(* Logix 5000 project; controller IF2_DEMO Emulate 5570 rev 20.12; software revision 20.04; part 7 of 8 *)
(* tags used below, declared in another part *)
   Alarm_Packer1_Blocked : ALARM_DIGITAL;
   Alarm_Packer1_Starved : ALARM_DIGITAL;
   Alarm_Packer1_Stopped : ALARM_DIGITAL;
   Current_OEE_Availability : REAL;
   Current_OEE_Availability_MUL100 : DINT;
   Current_OEE_Available : REAL;
   Current_OEE_AvailableTimer : TIMER;
   Current_OEE_Overall : REAL;
   Current_OEE_Performance : REAL;
   Current_OEE_Performance_MUL100 : DINT;
   Current_OEE_Quality : REAL;
   Current_OEE_Quality_MUL100 : DINT;
   Current_OEE_Running : REAL;
   Current_OEE_RunningTimer : TIMER;
   OEE_Availability_Previous_1 : REAL;
   OEE_Availability_Previous_2 : REAL;
   OEE_Availability_Previous_3 : REAL;
   OEE_Overall_Previous_1 : REAL;
   OEE_Overall_Previous_2 : REAL;
   OEE_Overall_Previous_3 : REAL;
   OEE_Performance_Previous_1 : REAL;
   OEE_Performance_Previous_2 : REAL;
   OEE_Performance_Previous_3 : REAL;
   OEE_Quality_Previous_1 : REAL;
   OEE_Quality_Previous_2 : REAL;
   OEE_Quality_Previous_3 : REAL;
   OutputTargetTimer : TIMER;
   Packaging_Cases_Good : DINT;
   Packaging_Cases_Per_Minute : REAL;
   Packaging_Cases_Rejected : DINT;
   Packaging_Cases_Total : DINT;
   Packaging_Status : DINT;
   Packer : FTVPDemoWorkCell;
   Packer_State : DINT;
   TempReadTrigger : TIMER;
   TempTimer : TIMER;
   TempTimer2 : TIMER;
   ChangeOver_In_Progress : BOOL;
   Current_Order : STRING;
   CurrentCustomerName : STRING;
   CurrentPartName : STRING;
   IF_OEE : IF_OEE;
   InstantFizz_Plant : Plant;
   Line1 : FTVPDemoLine;
   Line_State_String : State;
   LineStates : STRING[4];
   NewOrder_Trigger : Event_Triggers;
   OEE_Part_Scrap_Old : DINT;
   OEE_Parts_Good_Old : DINT;
   OEE_Parts_Total_Old : DINT;
   OEE_Scrap_Filler : DINT;
   OEE_Scrap_Labeler : DINT;
   OEE_Scrap_Packaging : DINT;
   OrderQty : DINT[4];
   PartCountRollOver : DINT;
   Performance_Control : DINT;
   Previous_Order : STRING;
   PreviousCustomerName : STRING;
   PreviousPartName : STRING;
   ProdCounts : Counts;
   Timer1000ms : TIMER;
   Timer250ms : TIMER;
   WallClock : DINT[7];
   WC : WC[10];
(* PackD, continued *)

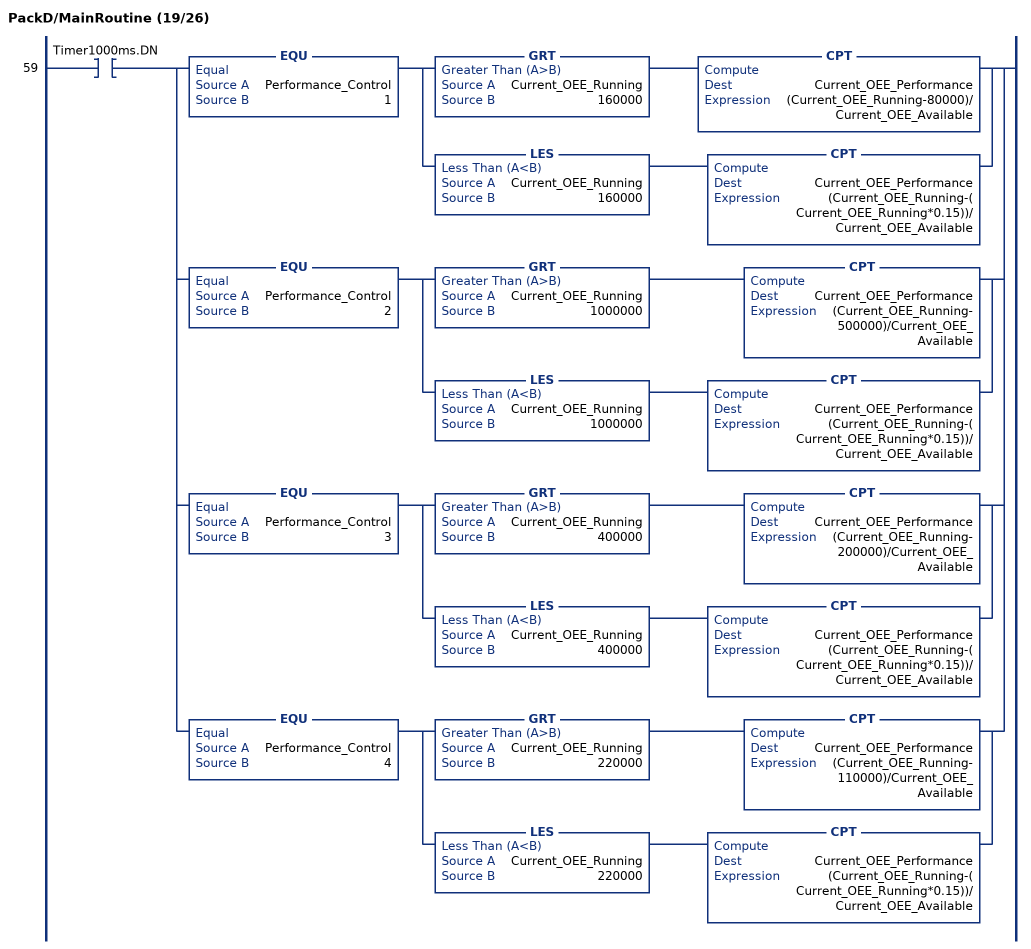
   59: XIC(Timer1000ms.DN)[EQU(Performance_Control,1) [GRT(Current_OEE_Running,160000) CPT(Current_OEE_Performance,(Current_OEE_Running-80000)/Current_OEE_Available) ,LES(Current_OEE_Running,160000) CPT(Current_OEE_Performance,(Current_OEE_Running-(Current_OEE_Running*0.15))/Current_OEE_Available) ] ,EQU(Performance_Control,2) [GRT(Current_OEE_Running,1000000) CPT(Current_OEE_Performance,(Current_OEE_Running-500000)/Current_OEE_Available) ,LES(Current_OEE_Running,1000000) CPT(Current_OEE_Performance,(Current_OEE_Running-(Current_OEE_Running*0.15))/Current_OEE_Available) ] ,EQU(Performance_Control,3) [GRT(Current_OEE_Running,400000) CPT(Current_OEE_Performance,(Current_OEE_Running-200000)/Current_OEE_Available) ,LES(Current_OEE_Running,400000) CPT(Current_OEE_Performance,(Current_OEE_Running-(Current_OEE_Running*0.15))/Current_OEE_Available) ] ,EQU(Performance_Control,4) [GRT(Current_OEE_Running,220000) CPT(Current_OEE_Performance,(Current_OEE_Running-110000)/Current_OEE_Available) ,LES(Current_OEE_Running,220000) CPT(Current_OEE_Performance,(Current_OEE_Running-(Current_OEE_Running*0.15))/Current_OEE_Available) ] ];
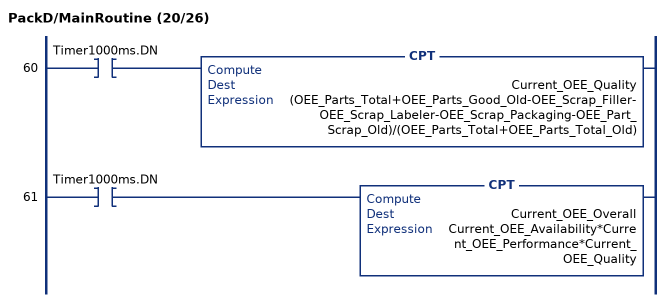
   60: XIC(Timer1000ms.DN)CPT(Current_OEE_Quality,(OEE_Parts_Total+OEE_Parts_Good_Old-OEE_Scrap_Filler-OEE_Scrap_Labeler-OEE_Scrap_Packaging-OEE_Part_Scrap_Old)/(OEE_Parts_Total+OEE_Parts_Total_Old));
   61: XIC(Timer1000ms.DN)CPT(Current_OEE_Overall,Current_OEE_Availability*Current_OEE_Performance*Current_OEE_Quality);
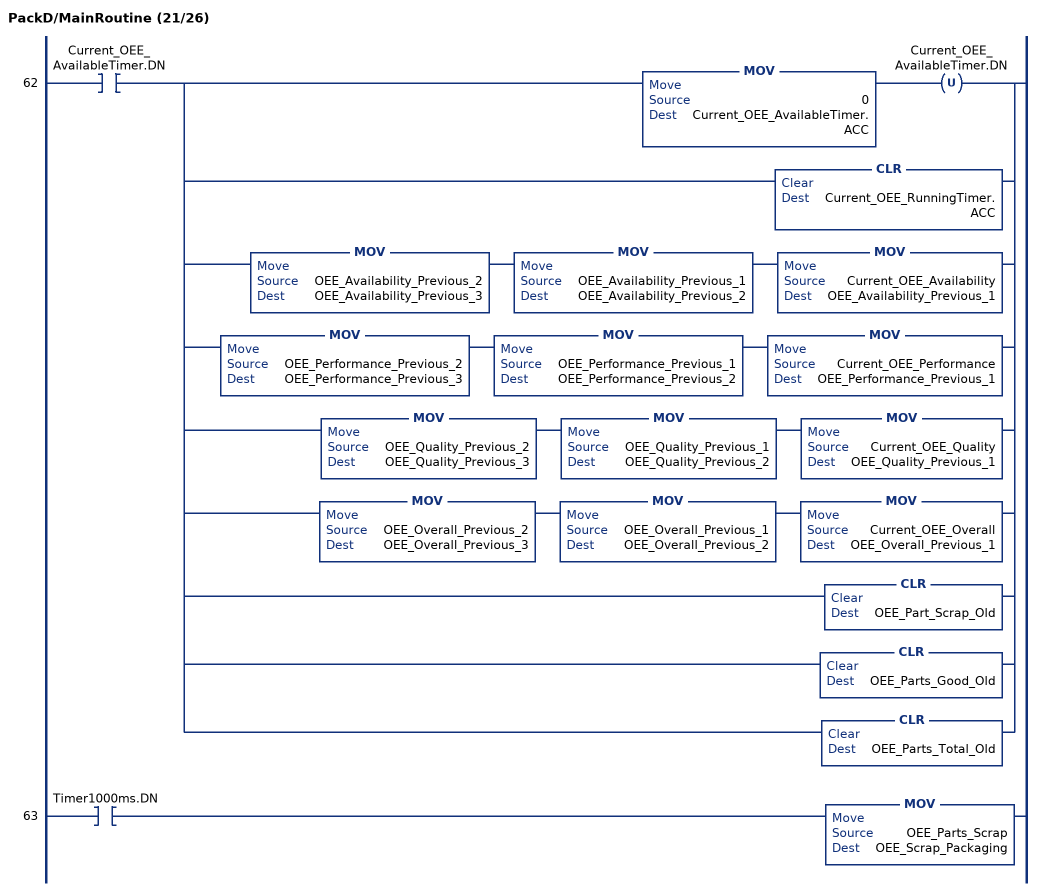
   62: XIC(Current_OEE_AvailableTimer.DN)[MOV(0,Current_OEE_AvailableTimer.ACC) OTU(Current_OEE_AvailableTimer.DN) ,CLR(Current_OEE_RunningTimer.ACC) ,MOV(OEE_Availability_Previous_2,OEE_Availability_Previous_3) MOV(OEE_Availability_Previous_1,OEE_Availability_Previous_2) MOV(Current_OEE_Availability,OEE_Availability_Previous_1) ,MOV(OEE_Performance_Previous_2,OEE_Performance_Previous_3) MOV(OEE_Performance_Previous_1,OEE_Performance_Previous_2) MOV(Current_OEE_Performance,OEE_Performance_Previous_1) ,MOV(OEE_Quality_Previous_2,OEE_Quality_Previous_3) MOV(OEE_Quality_Previous_1,OEE_Quality_Previous_2) MOV(Current_OEE_Quality,OEE_Quality_Previous_1) ,MOV(OEE_Overall_Previous_2,OEE_Overall_Previous_3) MOV(OEE_Overall_Previous_1,OEE_Overall_Previous_2) MOV(Current_OEE_Overall,OEE_Overall_Previous_1) ,CLR(OEE_Part_Scrap_Old) ,CLR(OEE_Parts_Good_Old) ,CLR(OEE_Parts_Total_Old) ];
   63: XIC(Timer1000ms.DN)MOV(OEE_Parts_Scrap,OEE_Scrap_Packaging);
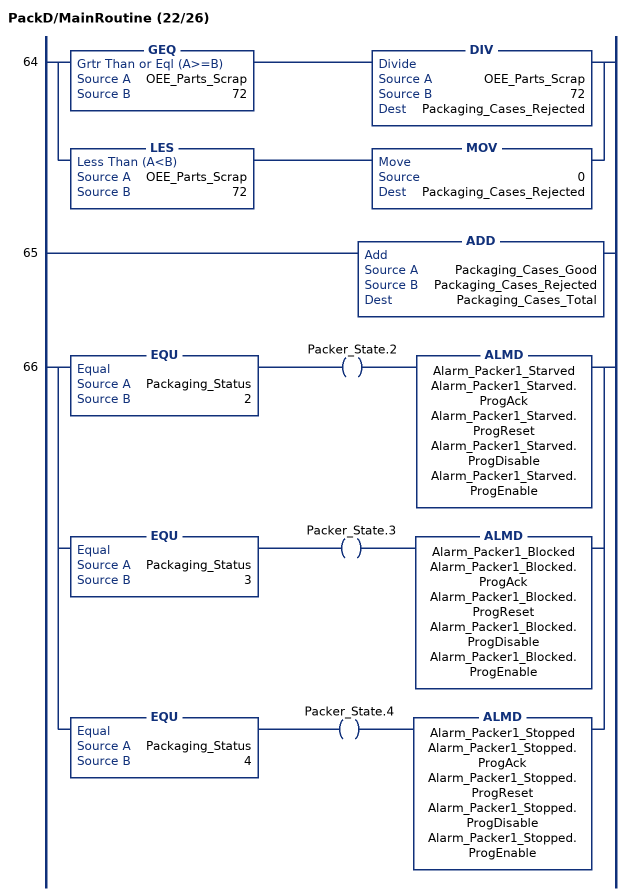
   64: [GEQ(OEE_Parts_Scrap,72) DIV(OEE_Parts_Scrap,72,Packaging_Cases_Rejected) ,LES(OEE_Parts_Scrap,72) MOV(0,Packaging_Cases_Rejected) ];
   65: ADD(Packaging_Cases_Good,Packaging_Cases_Rejected,Packaging_Cases_Total);
   66: [EQU(Packaging_Status,2) OTE(Packer_State.2) ALMD(Alarm_Packer1_Starved,Alarm_Packer1_Starved.ProgAck,Alarm_Packer1_Starved.ProgReset,Alarm_Packer1_Starved.ProgDisable,Alarm_Packer1_Starved.ProgEnable) ,EQU(Packaging_Status,3) OTE(Packer_State.3) ALMD(Alarm_Packer1_Blocked,Alarm_Packer1_Blocked.ProgAck,Alarm_Packer1_Blocked.ProgReset,Alarm_Packer1_Blocked.ProgDisable,Alarm_Packer1_Blocked.ProgEnable) ,EQU(Packaging_Status,4) OTE(Packer_State.4) ALMD(Alarm_Packer1_Stopped,Alarm_Packer1_Stopped.ProgAck,Alarm_Packer1_Stopped.ProgReset,Alarm_Packer1_Stopped.ProgDisable,Alarm_Packer1_Stopped.ProgEnable) ];
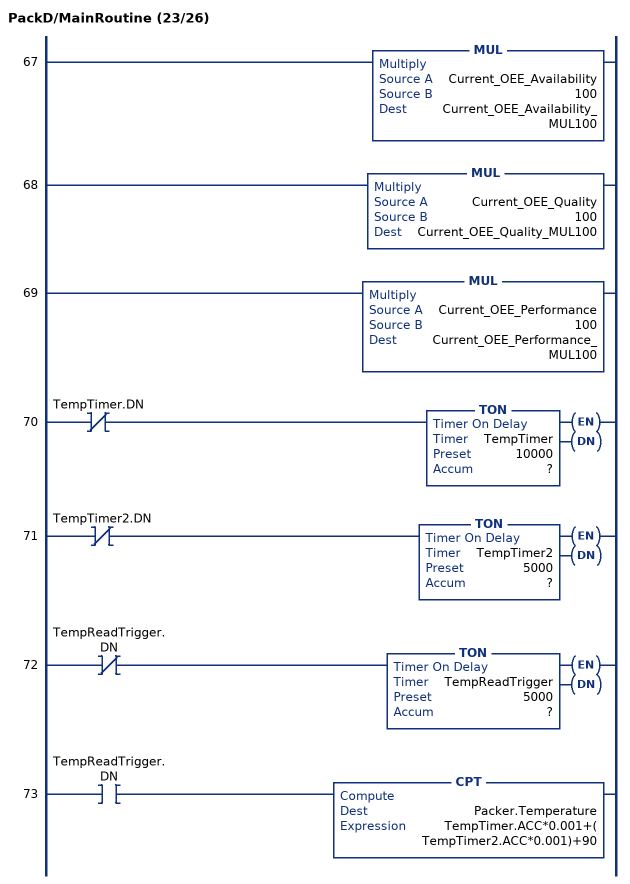
   67: MUL(Current_OEE_Availability,100,Current_OEE_Availability_MUL100);
   68: MUL(Current_OEE_Quality,100,Current_OEE_Quality_MUL100);
   69: MUL(Current_OEE_Performance,100,Current_OEE_Performance_MUL100);
   70: XIO(TempTimer.DN)TON(TempTimer,?,?);
   71: XIO(TempTimer2.DN)TON(TempTimer2,?,?);
   72: XIO(TempReadTrigger.DN)TON(TempReadTrigger,?,?);
   73: XIC(TempReadTrigger.DN)CPT(Packer.Temperature,TempTimer.ACC*0.001+(TempTimer2.ACC*0.001)+90);
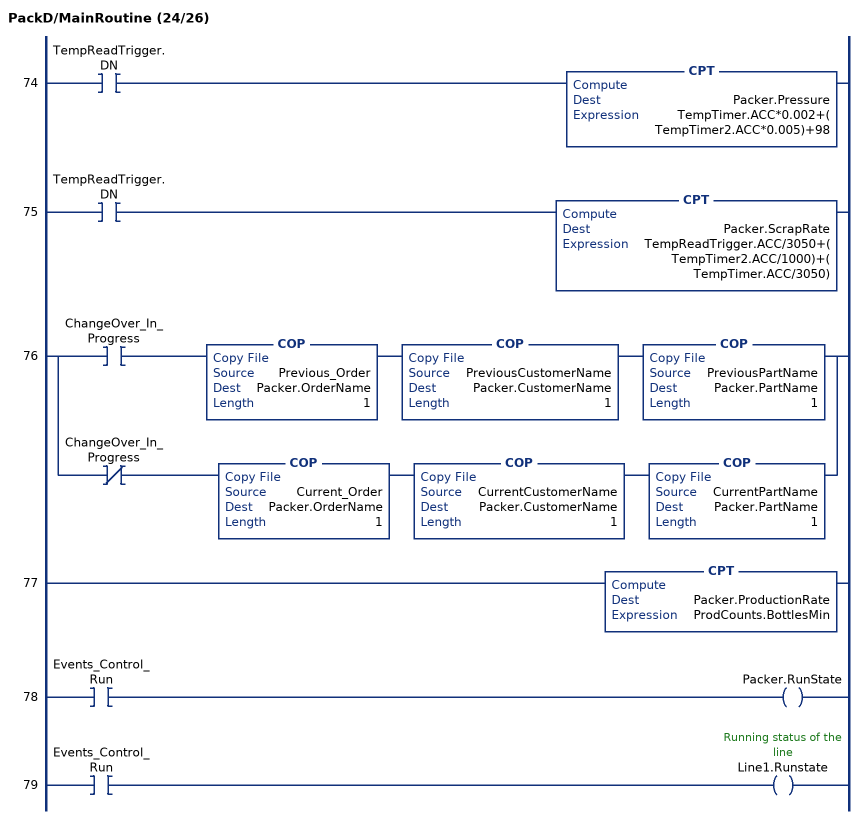
   74: XIC(TempReadTrigger.DN)CPT(Packer.Pressure,TempTimer.ACC*0.002+(TempTimer2.ACC*0.005)+98);
   75: XIC(TempReadTrigger.DN)CPT(Packer.ScrapRate,TempReadTrigger.ACC/3050+(TempTimer2.ACC/1000)+(TempTimer.ACC/3050));
   76: [XIC(ChangeOver_In_Progress) COP(Previous_Order,Packer.OrderName,1) COP(PreviousCustomerName,Packer.CustomerName,1) COP(PreviousPartName,Packer.PartName,1) ,XIO(ChangeOver_In_Progress) COP(Current_Order,Packer.OrderName,1) COP(CurrentCustomerName,Packer.CustomerName,1) COP(CurrentPartName,Packer.PartName,1) ];
   77: CPT(Packer.ProductionRate,ProdCounts.BottlesMin);
   78: XIC(Events_Control_Run)OTE(Packer.RunState);
   79: XIC(Events_Control_Run)OTE(Line1.Runstate);
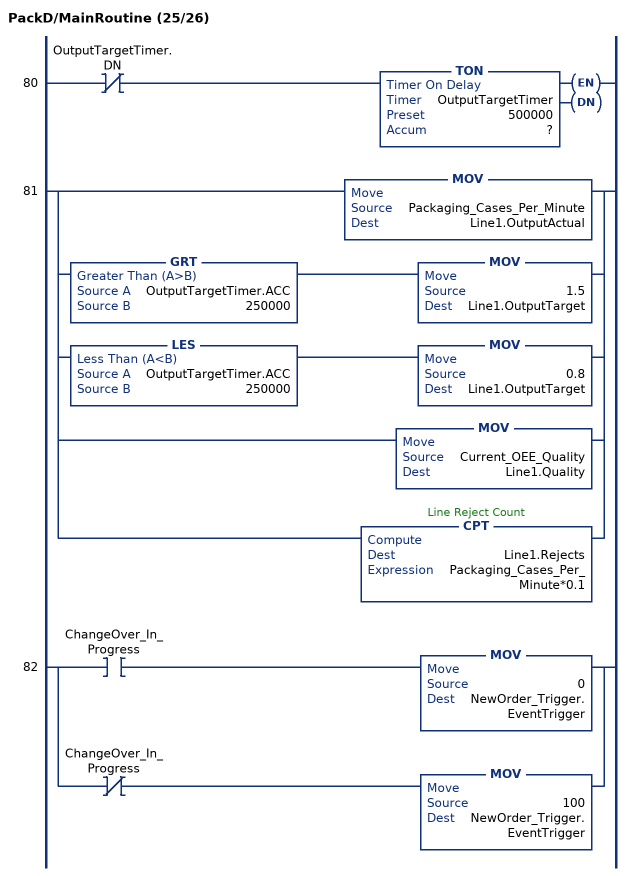
   80: XIO(OutputTargetTimer.DN)TON(OutputTargetTimer,?,?);
   81: [MOV(Packaging_Cases_Per_Minute,Line1.OutputActual) ,[GRT(OutputTargetTimer.ACC,250000) MOV(1.5,Line1.OutputTarget) ,LES(OutputTargetTimer.ACC,250000) MOV(0.8,Line1.OutputTarget) ] ,MOV(Current_OEE_Quality,Line1.Quality) ,CPT(Line1.Rejects,Packaging_Cases_Per_Minute*0.1) ];
   82: [XIC(ChangeOver_In_Progress) MOV(0,NewOrder_Trigger.EventTrigger) ,XIO(ChangeOver_In_Progress) MOV(100,NewOrder_Trigger.EventTrigger) ];
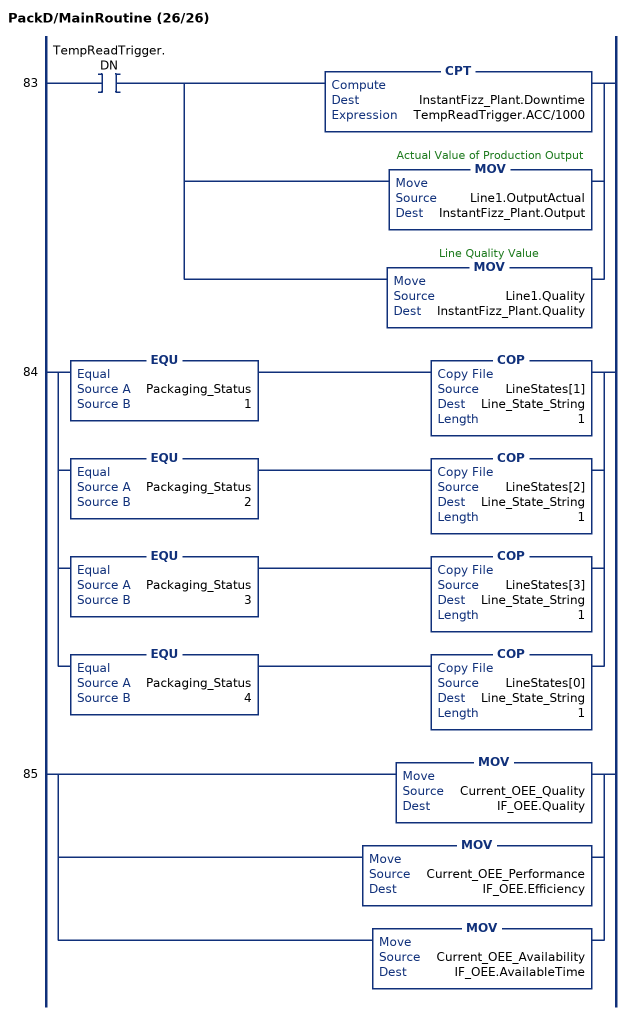
   83: XIC(TempReadTrigger.DN)[CPT(InstantFizz_Plant.Downtime,TempReadTrigger.ACC/1000) ,MOV(Line1.OutputActual,InstantFizz_Plant.Output) ,MOV(Line1.Quality,InstantFizz_Plant.Quality) ];
   84: [EQU(Packaging_Status,1) COP(LineStates[1],Line_State_String,1) ,EQU(Packaging_Status,2) COP(LineStates[2],Line_State_String,1) ,EQU(Packaging_Status,3) COP(LineStates[3],Line_State_String,1) ,EQU(Packaging_Status,4) COP(LineStates[0],Line_State_String,1) ];
   85: [MOV(Current_OEE_Quality,IF_OEE.Quality) ,MOV(Current_OEE_Performance,IF_OEE.Efficiency) ,MOV(Current_OEE_Availability,IF_OEE.AvailableTime) ];
END_ROUTINE
END_PROGRAM

PROGRAM Packer1   (* main routine MainRoutine *)
VAR
   Auto_setpoint : DINT := 3;
   Blinker : TIMER := (PRE := 1000, ACC := 931, EN := 1, TT := 1);
   Blocked_L : BOOL;
   Bottle_count_switch : BOOL := 1;
   Bottle_Counter : COUNTER := (ACC := 5098, CU := 1, DN := 1);
   BTank1_heat_ON : BOOL := 1;   // start heating
   BTank2_heat_ON : BOOL := 1;
   BTank3_heat_ON : BOOL := 1;
   BTMTimer_BTank1 : TIMER := (PRE := 1, EN := 1, TT := 1);   // Batch Tank1 timer
        .DN   // Batch Tank1 timer
   BTMTimer_BTank2 : TIMER := (PRE := 1, EN := 1, TT := 1);
   BTMTimer_BTank3 : TIMER := (PRE := 1, EN := 1, TT := 1);
   Drive_running : BOOL := 1;
   E_Stop : BOOL := 1;
   Events : Events := (Operate.OrderProc := 1, Control.StandbyCode := 3);
   Events_Control_Auto : ALIAS FOR WC_L.EventTrigger[0].5;
   Events_Control_Run : ALIAS FOR WC_L.EventTrigger[0].1;
   Events_Control_Standby : ALIAS FOR WC_L.EventTrigger[0].0;
   Events_Control_StandbyCode : ALIAS FOR WC_L.EventValue_REAL[1];
   Events_DownTime_Breakdown : ALIAS FOR WC_L.EventTrigger[0].2;
   Events_DownTime_BreakdownCode : ALIAS FOR WC_L.EventValue_REAL[2];
   Events_DownTime_Testing : ALIAS FOR WC_L.EventTrigger[0].7;
   Events_DownTime_UnschedMaint : ALIAS FOR WC_L.EventTrigger[0].6;
   Events_Operate_Load : ALIAS FOR WC_L.EventTrigger[0].10;
   Events_Operate_OrderProc : ALIAS FOR WC_L.EventTrigger[0].11;
   Events_Operate_Setup : ALIAS FOR WC_L.EventTrigger[0].9;
   Fill1_pressure : DINT := 150;   // Batch Tank1 pressure
   Fill2_pressure : DINT := 32;
   Fill3_pressure : DINT := 21;
   Heat_rate1 : REAL := 0.0003;   // value between 0 and 0.1
   Heat_rate2 : REAL := 0.0007;
   Heat_rate3 : REAL := 1.e-04;
   HMI : HMIVars := (ScrapRate := 5.0, SpeedControl := 100.0, PrevSpeed := 100.0, PartCountRollOver := 9999999, MfgTimeBase := 1, MaxEventDur := 19.0, MinEventDur := 6.0, EventsPerHr := 100, EventDur := 9.167803, RunDur := 25.832197, MinRunDur := 5.0);
   Jog : BOOL;
   Jog_PB : BOOL;
   Manual : BOOL;
   MaxPsiSP1 : DINT := 150;   // maximum pressure setpoint
   MaxPsiSP2 : DINT := 150;
   MaxPsiSP3 : DINT := 150;
   MaxTempSP1 : DINT := 220;   // maximum temperature set point
   MaxTempSP2 : DINT := 220;
   MaxTempSP3 : DINT := 220;
   MfgOrders : MfgOrders := (CustomerName := 'MRP', OrderName := 'Product B 1', GetNextOrder := 1, OrderQty := 600, ProdRate := 11.0, SetupTime := 8.0, PartName := 'Bottle3', WorkcellName := 'Capper 3', OperationId := 1006558);
   MfgOrders_CustomerName : ALIAS FOR WC_L.FlexSTRING[4];
   MfgOrders_OrderName : ALIAS FOR WC_L.FlexSTRING[3];
   MfgOrders_PartName : ALIAS FOR WC_L.FlexSTRING[0];
   MinPsiSP1 : DINT;   // minimum pressure setpoint
   MinPsiSP2 : DINT;
   MinPsiSP3 : DINT;
   MinTempSP1 : DINT := 60;   // minimum setpoint for temperature
   MinTempSP2 : DINT := 60;
   MinTempSP3 : DINT := 60;
   Motor1_temperature : DINT := 220;   // Motor1Temperature
   Motor2_temperature : DINT := 101;
   Motor3_temperature : DINT := 77;
   OEE : OEE := (IdealCycleTime := 5.0);
   OEE_IdealCycleTime : ALIAS FOR WC_L.IdealCT;
   OEE_Parts_Good : ALIAS FOR WC_L.GoodParts;
   OEE_Parts_Scrap : ALIAS FOR WC_L.ScrapParts;
   OEE_Parts_Total : ALIAS FOR WC_L.TotalParts;
   Run_PB : BOOL;
   Run_PL : BOOL := 1;
   Run_start_timer : TIMER := (PRE := 2000);
   Running : BOOL := 1;
   SIM : SimVars := (Run.PRE := 25832, Event.PRE := 9168, Setup.PRE := 6000, EventNumber := 7, UtilityBool[2] := 1);
        .UTILITYBOOL[2]   // First Scan Bit
   Sin_input_float1 : REAL := 1.667488;
   Sin_input_float2 : REAL := 5.7742753;
   Sin_input_float3 : REAL := 4.0464277;
   Speed_setpoint : DINT := 3;
   Starved_L : BOOL;
   Stop_PB : BOOL;
   Stop_PL : BOOL;
   Suppress : Events;
   WC_L : ALIAS FOR WC[6];
END_VAR

ROUTINE MainRoutine   (* ladder *)
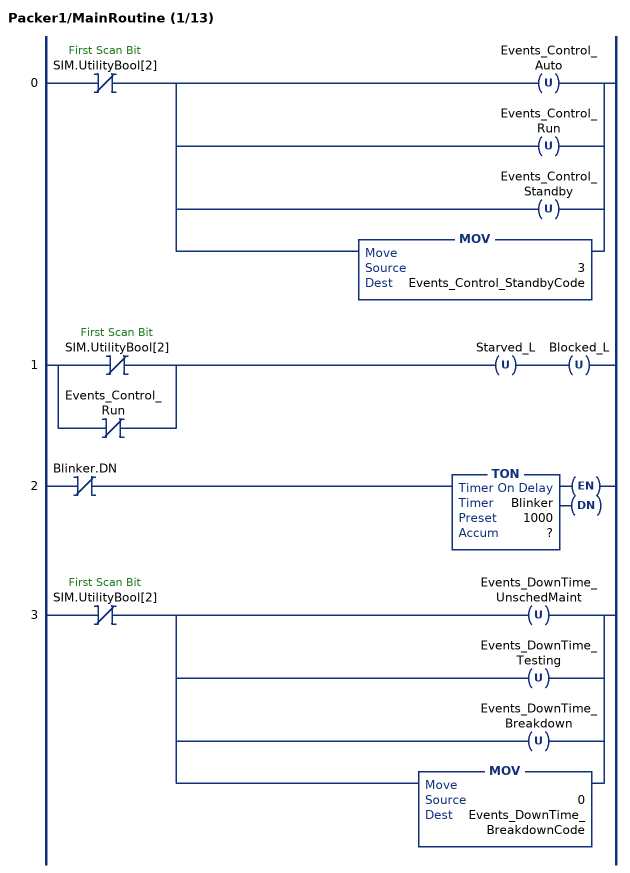
   0: XIO(SIM.UtilityBool[2])[OTU(Events_Control_Auto) ,OTU(Events_Control_Run) ,OTU(Events_Control_Standby) ,MOV(3,Events_Control_StandbyCode) ];
   1: [XIO(SIM.UtilityBool[2]) ,XIO(Events_Control_Run) ]OTU(Starved_L)OTU(Blocked_L);
   2: XIO(Blinker.DN)TON(Blinker,?,?);
   3: XIO(SIM.UtilityBool[2])[OTU(Events_DownTime_UnschedMaint) ,OTU(Events_DownTime_Testing) ,OTU(Events_DownTime_Breakdown) ,MOV(0,Events_DownTime_BreakdownCode) ];
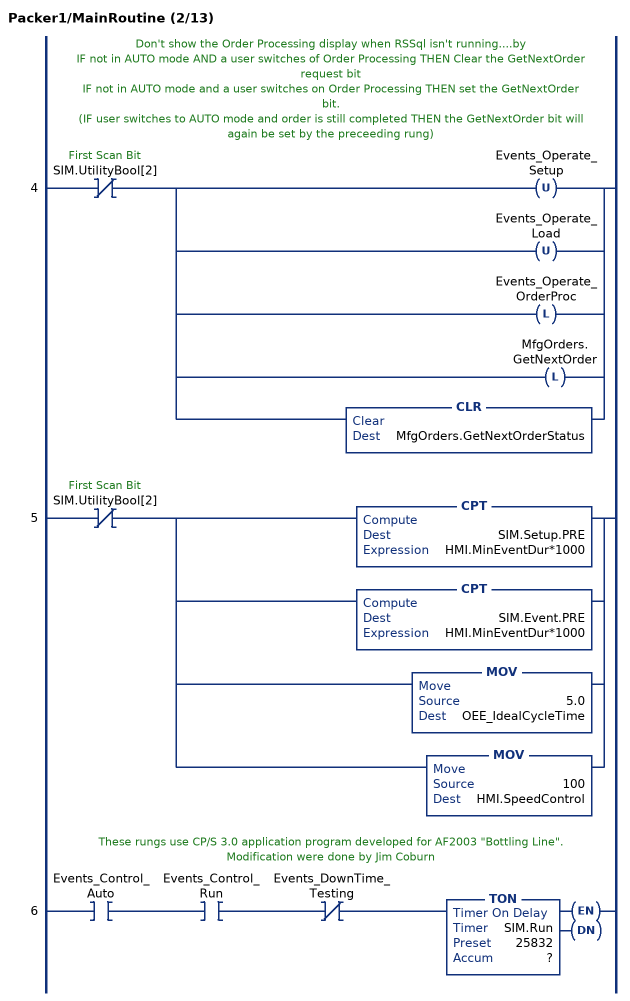
   // Don't show the Order Processing display when RSSql isn't running....by
   // IF not in AUTO mode AND a user switches of Order Processing THEN Clear the GetNextOrder request bit
   // IF not in AUTO mode and a user switches on Order Processing THEN set the GetNextOrder bit.
   // (IF user switches to AUTO mode and order is still completed THEN the GetNextOrder bit will again be set by the preceeding rung)
   4: XIO(SIM.UtilityBool[2])[OTU(Events_Operate_Setup) ,OTU(Events_Operate_Load) ,OTL(Events_Operate_OrderProc) ,OTL(MfgOrders.GetNextOrder) ,CLR(MfgOrders.GetNextOrderStatus) ];
   5: XIO(SIM.UtilityBool[2])[CPT(SIM.Setup.PRE,HMI.MinEventDur*1000) ,CPT(SIM.Event.PRE,HMI.MinEventDur*1000) ,MOV(5.0,OEE_IdealCycleTime) ,MOV(100,HMI.SpeedControl) ];
   // These rungs use CP/S 3.0 application program developed for AF2003 "Bottling Line".
   // Modification were done by Jim Coburn
   6: XIC(Events_Control_Auto)XIC(Events_Control_Run)XIO(Events_DownTime_Testing)TON(SIM.Run,?,?);
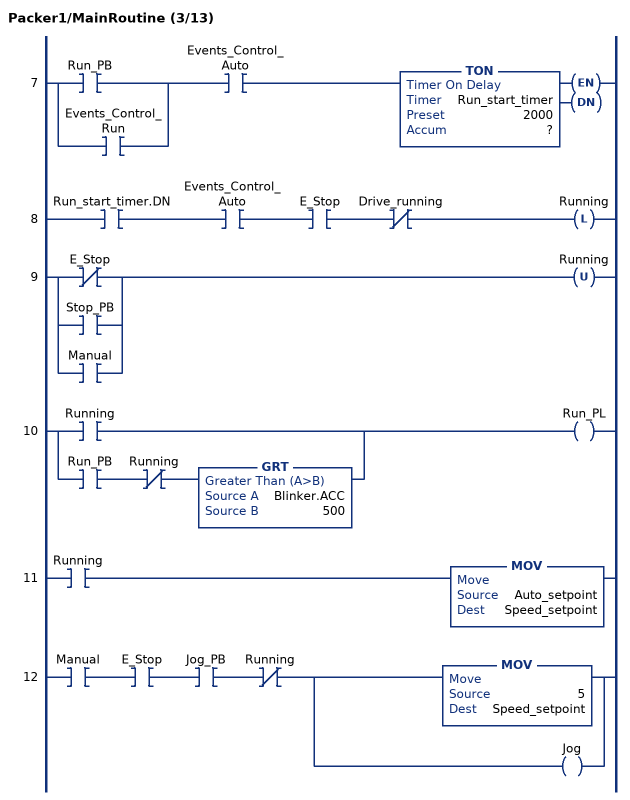
   7: [XIC(Run_PB) ,XIC(Events_Control_Run) ]XIC(Events_Control_Auto)TON(Run_start_timer,?,?);
   8: XIC(Run_start_timer.DN)XIC(Events_Control_Auto)XIC(E_Stop)XIO(Drive_running)OTL(Running);
   9: [XIO(E_Stop) ,[XIC(Stop_PB) ,XIC(Manual) ] ]OTU(Running);
   10: [XIC(Running) ,XIC(Run_PB) XIO(Running) GRT(Blinker.ACC,500) ]OTE(Run_PL);
   11: XIC(Running)MOV(Auto_setpoint,Speed_setpoint);
   12: XIC(Manual)XIC(E_Stop)XIC(Jog_PB)XIO(Running)[MOV(5,Speed_setpoint) ,OTE(Jog) ];
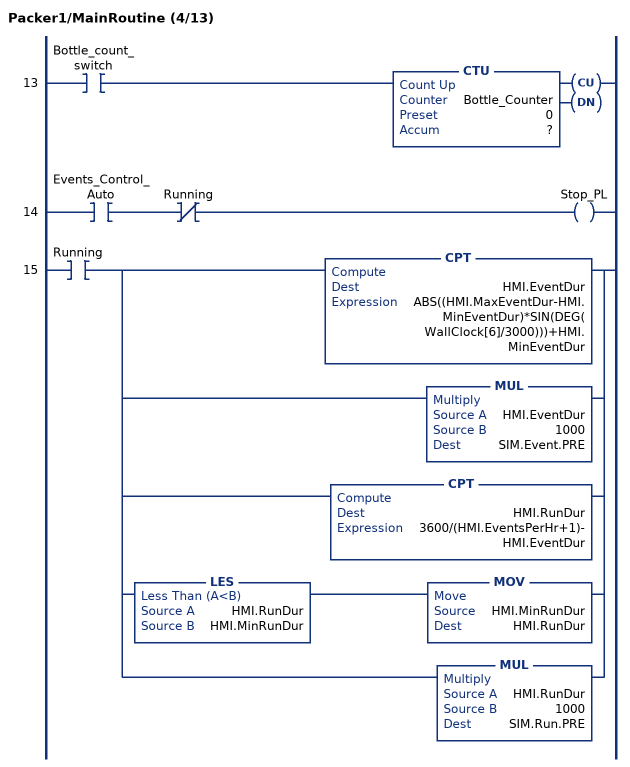
   13: XIC(Bottle_count_switch)CTU(Bottle_Counter,?,?);
   14: XIC(Events_Control_Auto)XIO(Running)OTE(Stop_PL);
   15: XIC(Running)[CPT(HMI.EventDur,ABS((HMI.MaxEventDur-HMI.MinEventDur)*SIN(DEG(WallClock[6]/3000)))+HMI.MinEventDur) ,MUL(HMI.EventDur,1000,SIM.Event.PRE) ,CPT(HMI.RunDur,3600/(HMI.EventsPerHr+1)-HMI.EventDur) ,LES(HMI.RunDur,HMI.MinRunDur) MOV(HMI.MinRunDur,HMI.RunDur) ,MUL(HMI.RunDur,1000,SIM.Run.PRE) ];
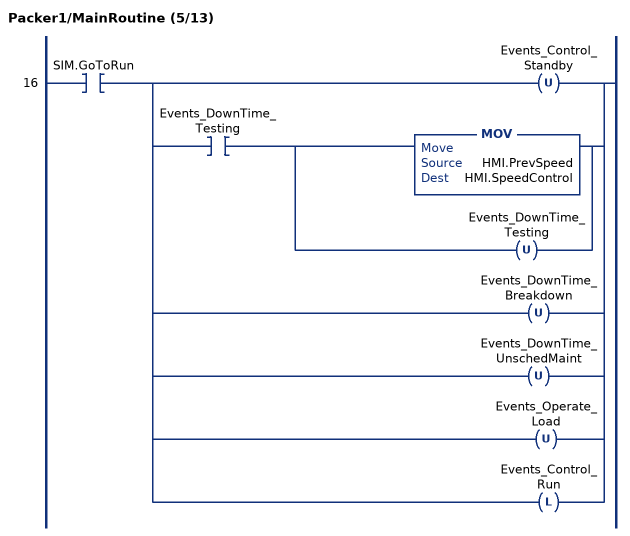
   16: XIC(SIM.GoToRun)[OTU(Events_Control_Standby) ,XIC(Events_DownTime_Testing) [MOV(HMI.PrevSpeed,HMI.SpeedControl) ,OTU(Events_DownTime_Testing) ] ,OTU(Events_DownTime_Breakdown) ,OTU(Events_DownTime_UnschedMaint) ,OTU(Events_Operate_Load) ,OTL(Events_Control_Run) ];
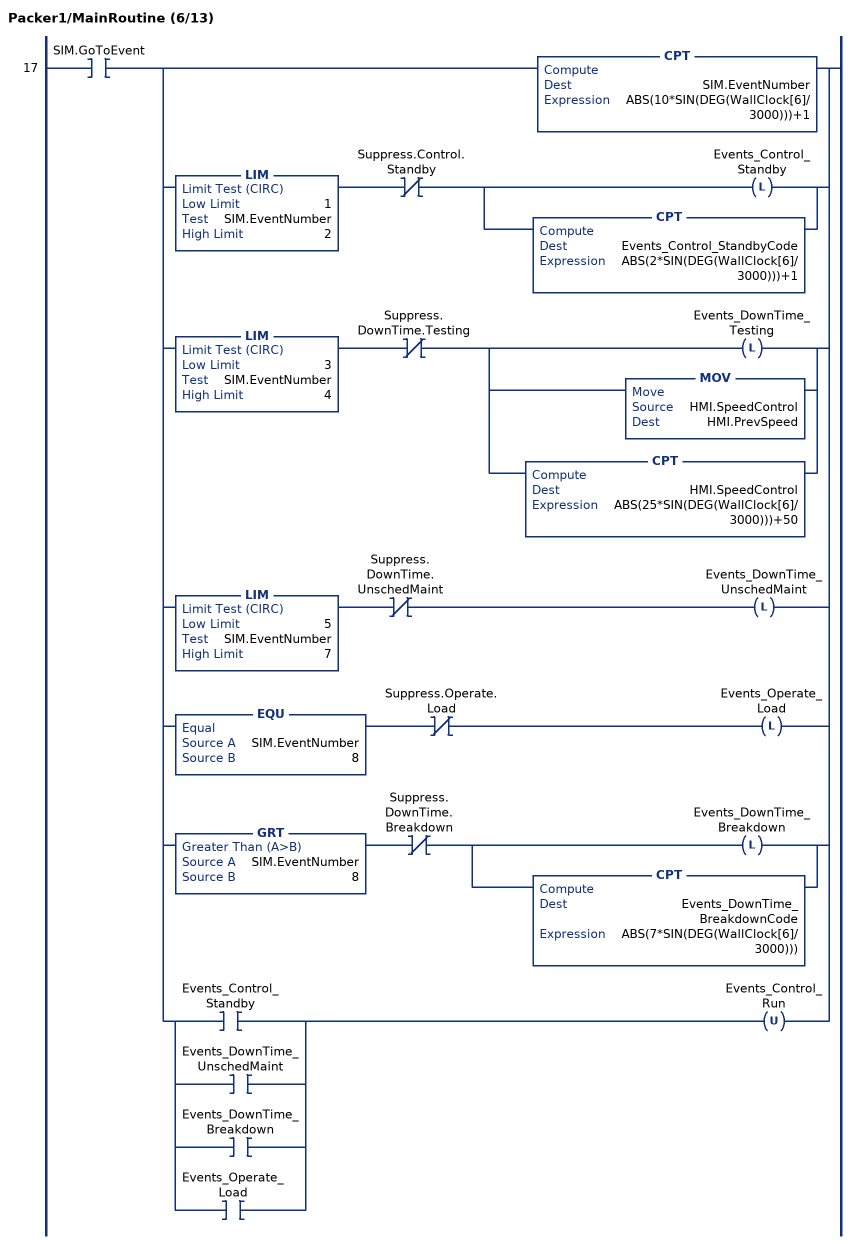
   17: XIC(SIM.GoToEvent)[CPT(SIM.EventNumber,ABS(10*SIN(DEG(WallClock[6]/3000)))+1) ,LIM(1,SIM.EventNumber,2) XIO(Suppress.Control.Standby) [OTL(Events_Control_Standby) ,CPT(Events_Control_StandbyCode,ABS(2*SIN(DEG(WallClock[6]/3000)))+1) ] ,LIM(3,SIM.EventNumber,4) XIO(Suppress.DownTime.Testing) [OTL(Events_DownTime_Testing) ,MOV(HMI.SpeedControl,HMI.PrevSpeed) ,CPT(HMI.SpeedControl,ABS(25*SIN(DEG(WallClock[6]/3000)))+50) ] ,LIM(5,SIM.EventNumber,7) XIO(Suppress.DownTime.UnschedMaint) OTL(Events_DownTime_UnschedMaint) ,EQU(SIM.EventNumber,8) XIO(Suppress.Operate.Load) OTL(Events_Operate_Load) ,GRT(SIM.EventNumber,8) XIO(Suppress.DownTime.Breakdown) [OTL(Events_DownTime_Breakdown) ,CPT(Events_DownTime_BreakdownCode,ABS(7*SIN(DEG(WallClock[6]/3000)))) ] ,[XIC(Events_Control_Standby) ,XIC(Events_DownTime_UnschedMaint) ,XIC(Events_DownTime_Breakdown) ,XIC(Events_Operate_Load) ] OTU(Events_Control_Run) ];
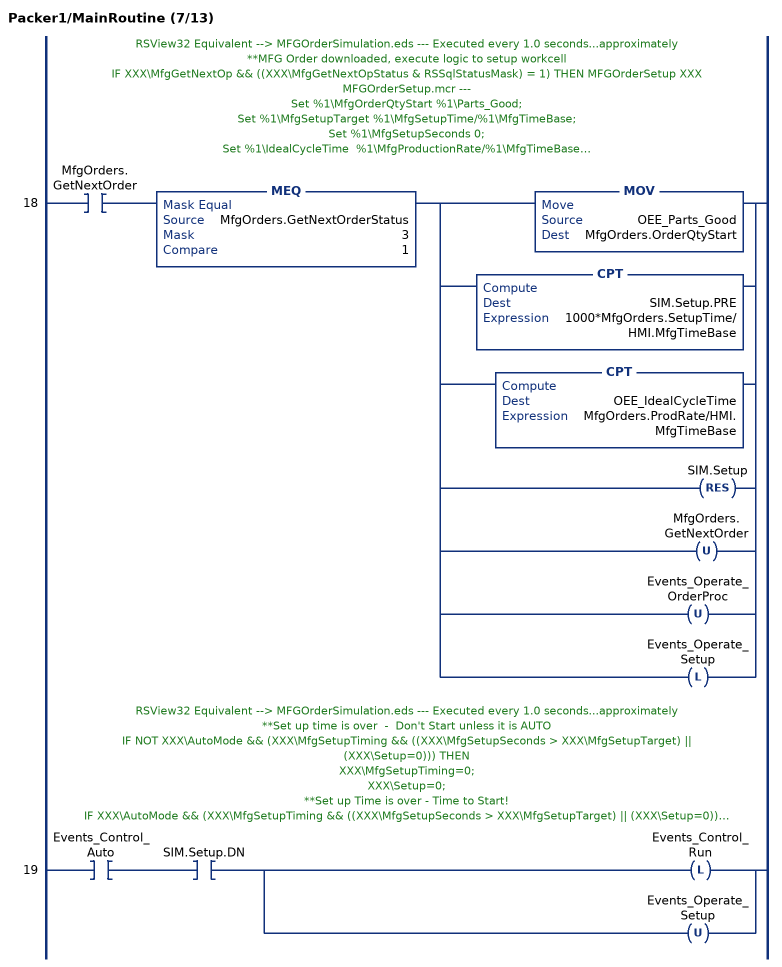
   // RSView32 Equivalent --> MFGOrderSimulation.eds --- Executed every 1.0 seconds...approximately
   // **MFG Order downloaded, execute logic to setup workcell
   // IF XXX\MfgGetNextOp && ((XXX\MfgGetNextOpStatus & RSSqlStatusMask) = 1) THEN MFGOrderSetup XXX
   // MFGOrderSetup.mcr ---
   // 	Set %1\MfgOrderQtyStart %1\Parts_Good;
   // 	Set %1\MfgSetupTarget %1\MfgSetupTime/%1\MfgTimeBase;
   // 	Set %1\MfgSetupSeconds 0;
   // 	Set %1\IdealCycleTime  %1\MfgProductionRate/%1\MfgTimeBase;
   // 	Set %1\MfgGetNextOp 0;
   // 	Set %1\Setup 1;
   // 	Set %1\OrderProcessing 0;
   // 	Set %1\MfgSetupTiming 1;
   18: XIC(MfgOrders.GetNextOrder)MEQ(MfgOrders.GetNextOrderStatus,3,1)[MOV(OEE_Parts_Good,MfgOrders.OrderQtyStart) ,CPT(SIM.Setup.PRE,1000*MfgOrders.SetupTime/HMI.MfgTimeBase) ,CPT(OEE_IdealCycleTime,MfgOrders.ProdRate/HMI.MfgTimeBase) ,RES(SIM.Setup) ,OTU(MfgOrders.GetNextOrder) ,OTU(Events_Operate_OrderProc) ,OTL(Events_Operate_Setup) ];
   // RSView32 Equivalent --> MFGOrderSimulation.eds --- Executed every 1.0 seconds...approximately
   // **Set up time is over  -  Don't Start unless it is AUTO
   // IF NOT XXX\AutoMode && (XXX\MfgSetupTiming && ((XXX\MfgSetupSeconds > XXX\MfgSetupTarget) || (XXX\Setup=0))) THEN
   // 	XXX\MfgSetupTiming=0;
   // 	XXX\Setup=0;
   // **Set up Time is over - Time to Start!
   // IF XXX\AutoMode && (XXX\MfgSetupTiming && ((XXX\MfgSetupSeconds > XXX\MfgSetupTarget) || (XXX\Setup=0))) THEN
   // 	XXX\MfgSetupTiming=0;
   // 	XXX\Setup=0;
   // 	XXX\RUNNING=1
   19: XIC(Events_Control_Auto)XIC(SIM.Setup.DN)[OTL(Events_Control_Run) ,OTU(Events_Operate_Setup) ];
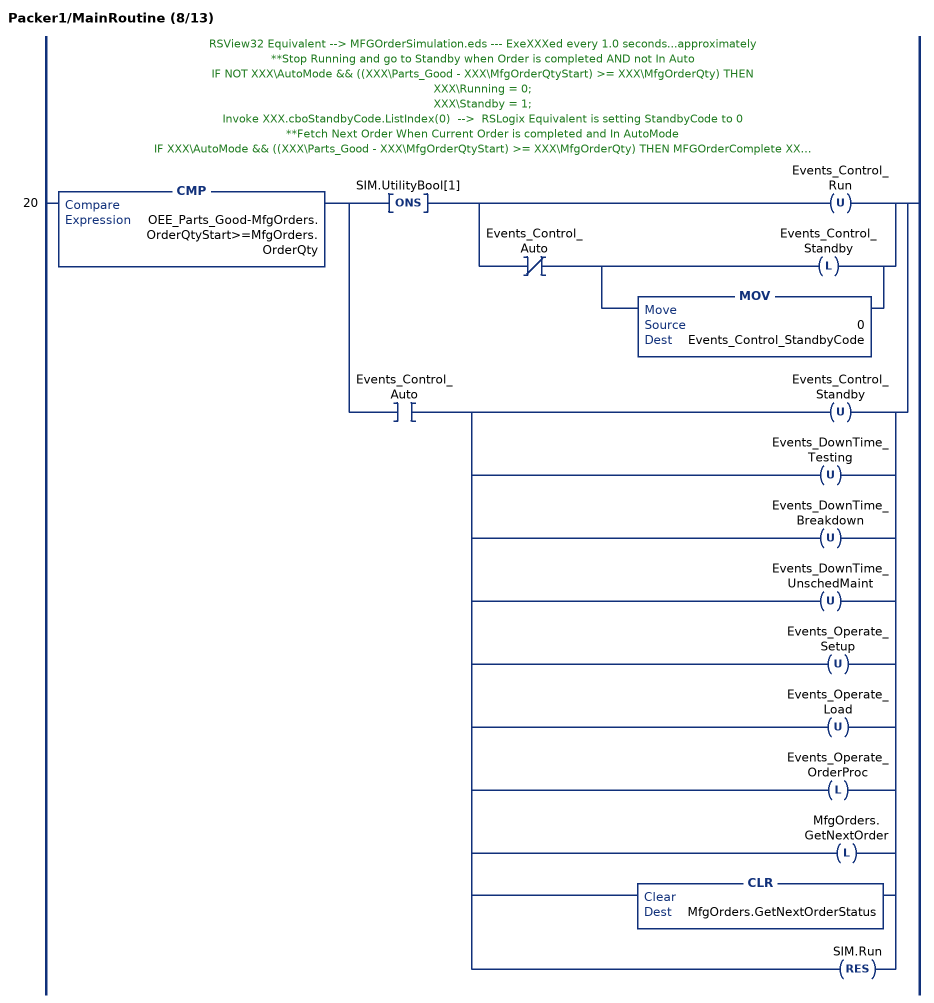
   // RSView32 Equivalent --> MFGOrderSimulation.eds --- ExeXXXed every 1.0 seconds...approximately
   // **Stop Running and go to Standby when Order is completed AND not In Auto
   // IF NOT XXX\AutoMode && ((XXX\Parts_Good - XXX\MfgOrderQtyStart) >= XXX\MfgOrderQty) THEN
   // 	XXX\Running = 0;
   // 	XXX\Standby = 1;
   // 	Invoke XXX.cboStandbyCode.ListIndex(0)  -->  RSLogix Equivalent is setting StandbyCode to 0
   // **Fetch Next Order When Current Order is completed and In AutoMode
   // IF XXX\AutoMode && ((XXX\Parts_Good - XXX\MfgOrderQtyStart) >= XXX\MfgOrderQty) THEN MFGOrderComplete XXX
   // MFGOrderComplete.mcr --- (Macros exeXXXed when called. %1 is the Workcell name -- typical all mcrs)
   // 	Set %1\RunStart %1\Timer;
   // 	Set %1\StandBy 0;
   // 	Set %1\Test 0;
   // 	Set %1\UnSchedMaint 0;
   // 	Set %1\Breakdown 0;
   // 	Set %1\Load 0;
   // 	Set %1\OrderProcessing 1;
   // 	Set %1\Running 0;
   // 	Set %1\MFGGetNextOpStatus 0;
   // 	Set %1\MFGGetNextOp 1
   20: CMP(OEE_Parts_Good-MfgOrders.OrderQtyStart>=MfgOrders.OrderQty)[ONS(SIM.UtilityBool[1]) [OTU(Events_Control_Run) ,XIO(Events_Control_Auto) [OTL(Events_Control_Standby) ,MOV(0,Events_Control_StandbyCode) ] ] ,XIC(Events_Control_Auto) [OTU(Events_Control_Standby) ,OTU(Events_DownTime_Testing) ,OTU(Events_DownTime_Breakdown) ,OTU(Events_DownTime_UnschedMaint) ,OTU(Events_Operate_Setup) ,OTU(Events_Operate_Load) ,OTL(Events_Operate_OrderProc) ,OTL(MfgOrders.GetNextOrder) ,CLR(MfgOrders.GetNextOrderStatus) ,RES(SIM.Run) ] ];
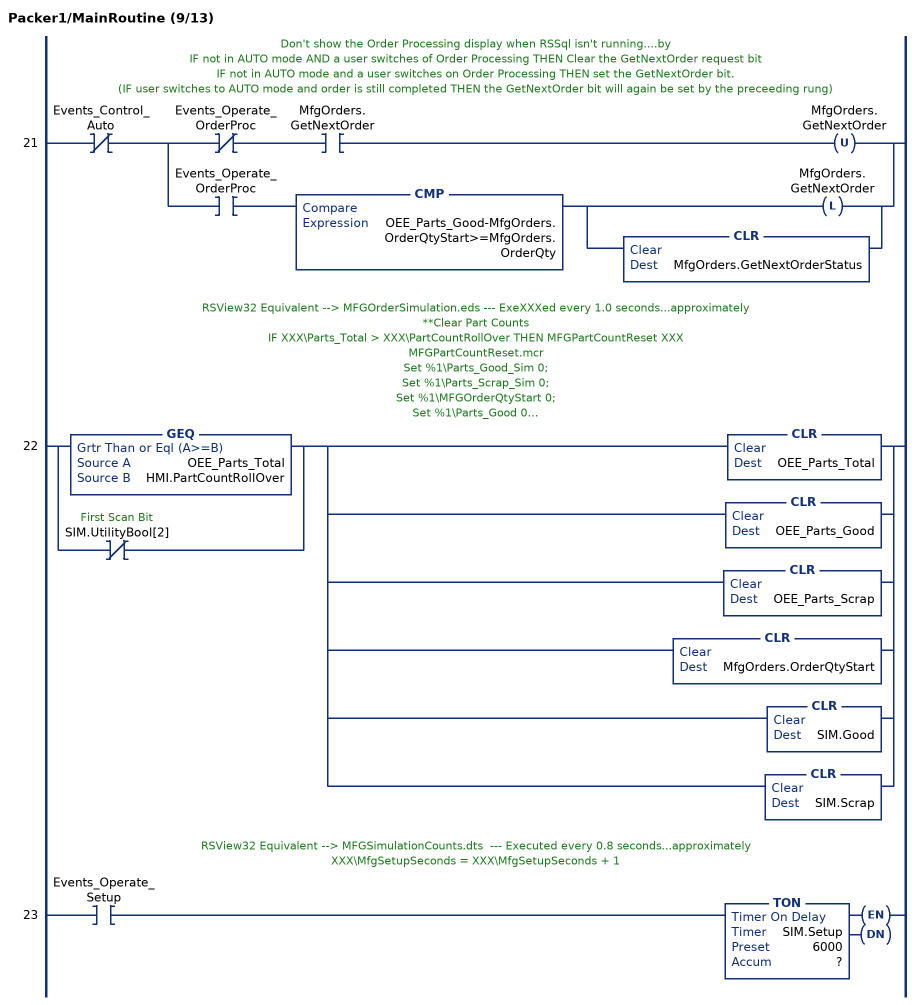
   // Don't show the Order Processing display when RSSql isn't running....by
   // IF not in AUTO mode AND a user switches of Order Processing THEN Clear the GetNextOrder request bit
   // IF not in AUTO mode and a user switches on Order Processing THEN set the GetNextOrder bit.
   // (IF user switches to AUTO mode and order is still completed THEN the GetNextOrder bit will again be set by the preceeding rung)
   21: XIO(Events_Control_Auto)[XIO(Events_Operate_OrderProc) XIC(MfgOrders.GetNextOrder) OTU(MfgOrders.GetNextOrder) ,XIC(Events_Operate_OrderProc) CMP(OEE_Parts_Good-MfgOrders.OrderQtyStart>=MfgOrders.OrderQty) [OTL(MfgOrders.GetNextOrder) ,CLR(MfgOrders.GetNextOrderStatus) ] ];
   // RSView32 Equivalent --> MFGOrderSimulation.eds --- ExeXXXed every 1.0 seconds...approximately
   // **Clear Part Counts
   // IF XXX\Parts_Total > XXX\PartCountRollOver THEN MFGPartCountReset XXX
   // MFGPartCountReset.mcr
   // 	Set %1\Parts_Good_Sim 0;
   // 	Set %1\Parts_Scrap_Sim 0;
   // 	Set %1\MFGOrderQtyStart 0;
   // 	Set %1\Parts_Good 0;
   // 	Set %1\Parts_Scrap 0;
   // 	Set %1\Parts_Total 0
   22: [GEQ(OEE_Parts_Total,HMI.PartCountRollOver) ,XIO(SIM.UtilityBool[2]) ][CLR(OEE_Parts_Total) ,CLR(OEE_Parts_Good) ,CLR(OEE_Parts_Scrap) ,CLR(MfgOrders.OrderQtyStart) ,CLR(SIM.Good) ,CLR(SIM.Scrap) ];
   // RSView32 Equivalent --> MFGSimulationCounts.dts	--- Executed every 0.8 seconds...approximately
   // XXX\MfgSetupSeconds = XXX\MfgSetupSeconds + 1
   23: XIC(Events_Operate_Setup)TON(SIM.Setup,?,?);
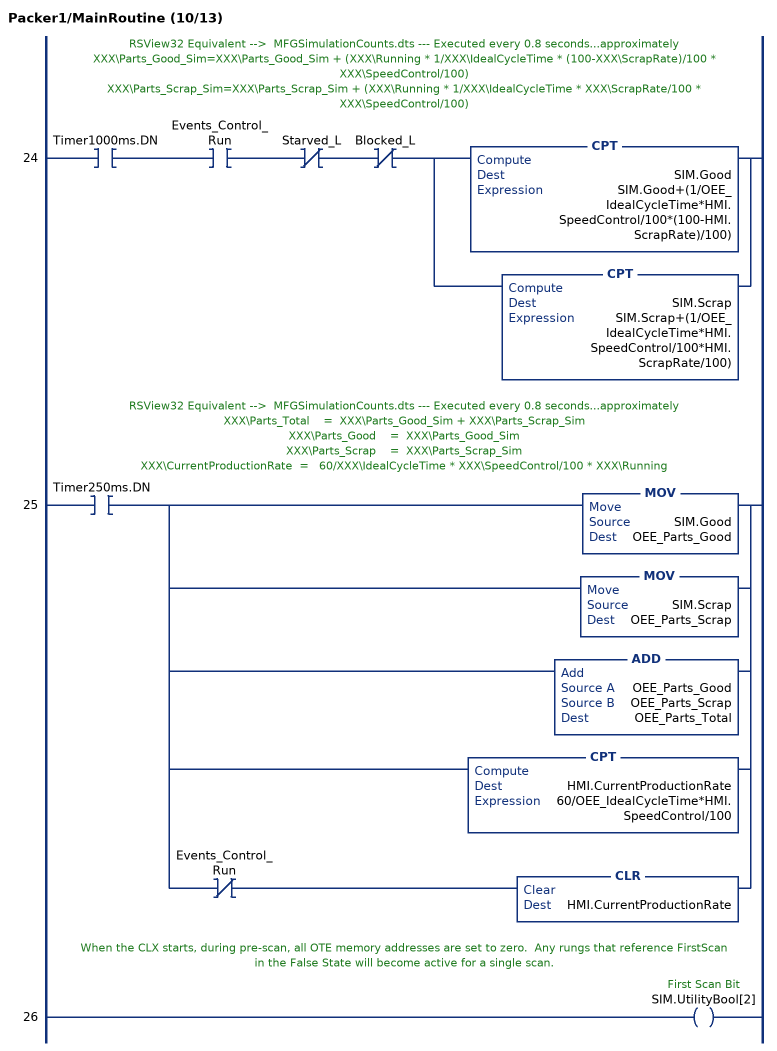
   // RSView32 Equivalent -->  MFGSimulationCounts.dts --- Executed every 0.8 seconds...approximately
   // XXX\Parts_Good_Sim=XXX\Parts_Good_Sim + (XXX\Running * 1/XXX\IdealCycleTime * (100-XXX\ScrapRate)/100 * XXX\SpeedControl/100)
   // XXX\Parts_Scrap_Sim=XXX\Parts_Scrap_Sim + (XXX\Running * 1/XXX\IdealCycleTime * XXX\ScrapRate/100 * XXX\SpeedControl/100)
   24: XIC(Timer1000ms.DN)XIC(Events_Control_Run)XIO(Starved_L)XIO(Blocked_L)[CPT(SIM.Good,SIM.Good+(1/OEE_IdealCycleTime*HMI.SpeedControl/100*(100-HMI.ScrapRate)/100)) ,CPT(SIM.Scrap,SIM.Scrap+(1/OEE_IdealCycleTime*HMI.SpeedControl/100*HMI.ScrapRate/100)) ];
   // RSView32 Equivalent -->  MFGSimulationCounts.dts --- Executed every 0.8 seconds...approximately
   // XXX\Parts_Total		=	XXX\Parts_Good_Sim + XXX\Parts_Scrap_Sim
   // XXX\Parts_Good		=	XXX\Parts_Good_Sim
   // XXX\Parts_Scrap		=	XXX\Parts_Scrap_Sim
   // XXX\CurrentProductionRate  = 	60/XXX\IdealCycleTime * XXX\SpeedControl/100 * XXX\Running
   25: XIC(Timer250ms.DN)[[MOV(SIM.Good,OEE_Parts_Good) ,MOV(SIM.Scrap,OEE_Parts_Scrap) ,ADD(OEE_Parts_Good,OEE_Parts_Scrap,OEE_Parts_Total) ] ,CPT(HMI.CurrentProductionRate,60/OEE_IdealCycleTime*HMI.SpeedControl/100) ,XIO(Events_Control_Run) CLR(HMI.CurrentProductionRate) ];
   // When the CLX starts, during pre-scan, all OTE memory addresses are set to zero.  Any rungs that reference FirstScan in the False State will become active for a single scan.
   26: OTE(SIM.UtilityBool[2]);
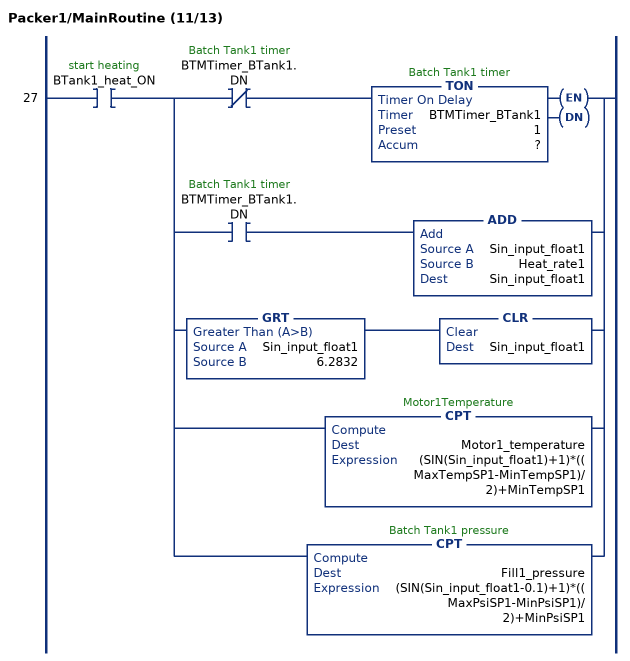
   27: XIC(BTank1_heat_ON)[XIO(BTMTimer_BTank1.DN) TON(BTMTimer_BTank1,?,?) ,XIC(BTMTimer_BTank1.DN) ADD(Sin_input_float1,Heat_rate1,Sin_input_float1) ,GRT(Sin_input_float1,6.2832) CLR(Sin_input_float1) ,[CPT(Motor1_temperature,(SIN(Sin_input_float1)+1)*((MaxTempSP1-MinTempSP1)/2)+MinTempSP1) ,CPT(Fill1_pressure,(SIN(Sin_input_float1-0.1)+1)*((MaxPsiSP1-MinPsiSP1)/2)+MinPsiSP1) ] ];
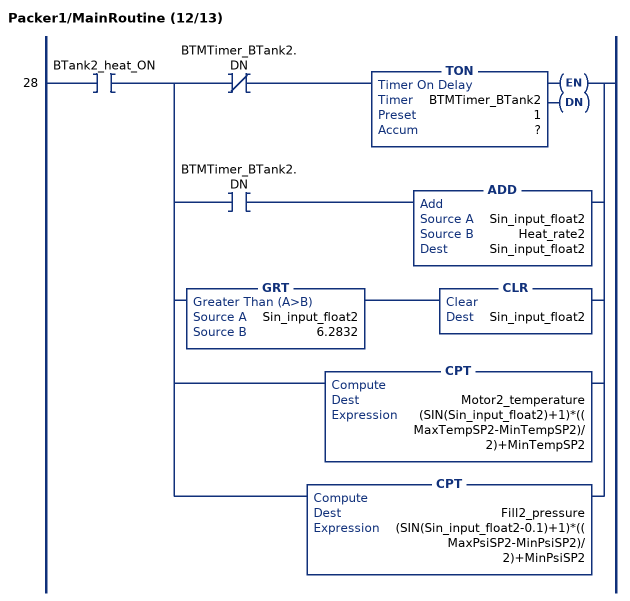
   28: XIC(BTank2_heat_ON)[XIO(BTMTimer_BTank2.DN) TON(BTMTimer_BTank2,?,?) ,XIC(BTMTimer_BTank2.DN) ADD(Sin_input_float2,Heat_rate2,Sin_input_float2) ,GRT(Sin_input_float2,6.2832) CLR(Sin_input_float2) ,[CPT(Motor2_temperature,(SIN(Sin_input_float2)+1)*((MaxTempSP2-MinTempSP2)/2)+MinTempSP2) ,CPT(Fill2_pressure,(SIN(Sin_input_float2-0.1)+1)*((MaxPsiSP2-MinPsiSP2)/2)+MinPsiSP2) ] ];
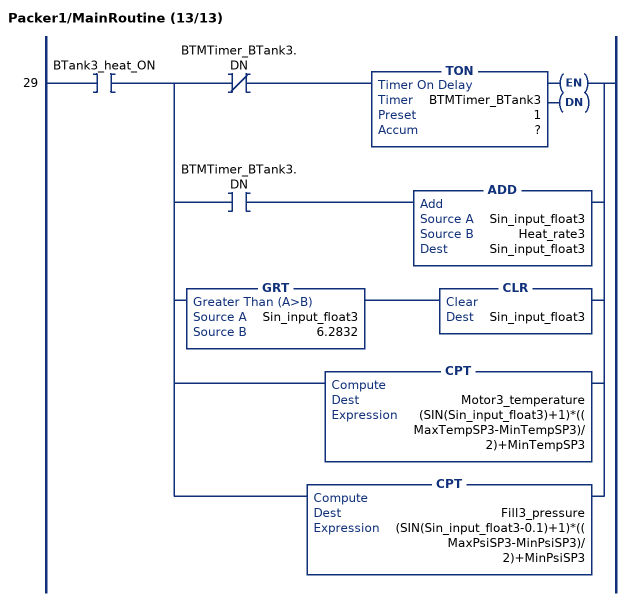
   29: XIC(BTank3_heat_ON)[XIO(BTMTimer_BTank3.DN) TON(BTMTimer_BTank3,?,?) ,XIC(BTMTimer_BTank3.DN) ADD(Sin_input_float3,Heat_rate3,Sin_input_float3) ,GRT(Sin_input_float3,6.2832) CLR(Sin_input_float3) ,[CPT(Motor3_temperature,(SIN(Sin_input_float3)+1)*((MaxTempSP3-MinTempSP3)/2)+MinTempSP3) ,CPT(Fill3_pressure,(SIN(Sin_input_float3-0.1)+1)*((MaxPsiSP3-MinPsiSP3)/2)+MinPsiSP3) ] ];
END_ROUTINE
END_PROGRAM
